{attribute 'linkalways'} 
{attribute 'no_explicit_call' := 'This FB is a CLASS and must be accessed using methods or properties'}
{attribute 'enable_dynamic_creation'}
FUNCTION_BLOCK Node_F_VN_ContourCircularityExp EXTENDS VisionNode
VAR
    ipContour : _ITcVnContainer;
    fCircularity : _LREAL(0.0);
    eMethod : _ETcVnCircularityCalculationMethod(ETcVnCircularityCalculationMethod.TCVN_CCM_DEFAULT);
    hrPrev : _HRESULT(S_OK);
	hresult : _HRESULT(S_OK);
END_VAR

METHOD PUBLIC  Clone : I_Node
VAR
	pNode : POINTER TO Node_F_VN_ContourCircularityExp;
END_VAR
pNode := __NEW(Node_F_VN_ContourCircularityExp);
Clone := pNode^;
END_METHOD

METHOD FB_init : BOOL
VAR_INPUT
	bInitRetains : BOOL; // if TRUE, the retain variables are initialized (warm start / cold start)
	bInCopyCode : BOOL;  // if TRUE, the instance afterwards gets moved into the copy code (online change)
END_VAR
AddInput('ipContour', ipContour);
AddParameter('eMethod', eMethod);
AddInput('hrPrev', hrPrev);
AddOutput('fCircularity', fCircularity);
AddOutput('hresult',hresult);
END_METHOD

METHOD PROTECTED OnExecute
hresult.Value := F_VN_ContourCircularityExp(
	ipContour := ipContour.Value,
    fCircularity := fCircularity.Value,
    eMethod := eMethod.Value,
	hrPrev:= hrPrev.Value);
END_METHOD

METHOD PUBLIC PreExecutionCheck
VAR_INPUT
	Check : I_PreExecutionChecks;
END_VAR
Check.IsTrue(ipContour.IsValid, 'ipContour must be a valid container');
Check.IsTrue((ipContour.IsType(TC_GLOBAL_CONST_LIST.ContainerType_Vector_TcVnPoint2_DINT) OR
              ipContour.IsType(TC_GLOBAL_CONST_LIST.ContainerType_Vector_TcVnPoint2_REAL)),
              'ipContour contains incorrect type');
END_METHOD

END_FUNCTION_BLOCK

(* stored: Version 1.1.0.1, ProductVersion 3.1.4026.13
   POU Node_F_VN_ContourCircularityExp: Id {628b586d-ab16-01fe-39d6-9190cd144228}, SpecialFunc None
   Folder Constructor: Id {24306136-84bf-0040-2e20-60610292534d}
   Method Clone: Id {d997facc-5961-004a-22e3-d5aa24fe1885}
   Method FB_init: Id {b91f812b-2927-0ba4-21f8-af1ff8ca408c}
   Method OnExecute: Id {6efb976b-defd-08f1-3b8e-8d39501889ac}
   Method PreExecutionCheck: Id {0a36e12f-f36d-0867-148f-b0bacab4f447} *)
